(* PLC project SafeLOGIC-1, BrAutomation SafeDESIGNER  5.15.0.0 *)
(* stored: companyURL http://www.br-automation.com, creationDateTime Sun Sep 18 11:29:32 2022 *)

PROGRAM Zone
  VAR  (* added by the conversion: wires and edge detectors of the diagram *)
    _SAFEBOOL_TO_BOOL243_OUT : BOOL;
    _SAFEBOOL_TO_BOOL256_OUT : BOOL;
    _AND_S244_OUT : ANY;
    _BOOL_TO_SAFEBOOL249_OUT : SAFEBOOL;
    _AND_S238_OUT : ANY;
    _OR259_OUT : BOOL;
    _AND246_OUT : BOOL;
  END_VAR

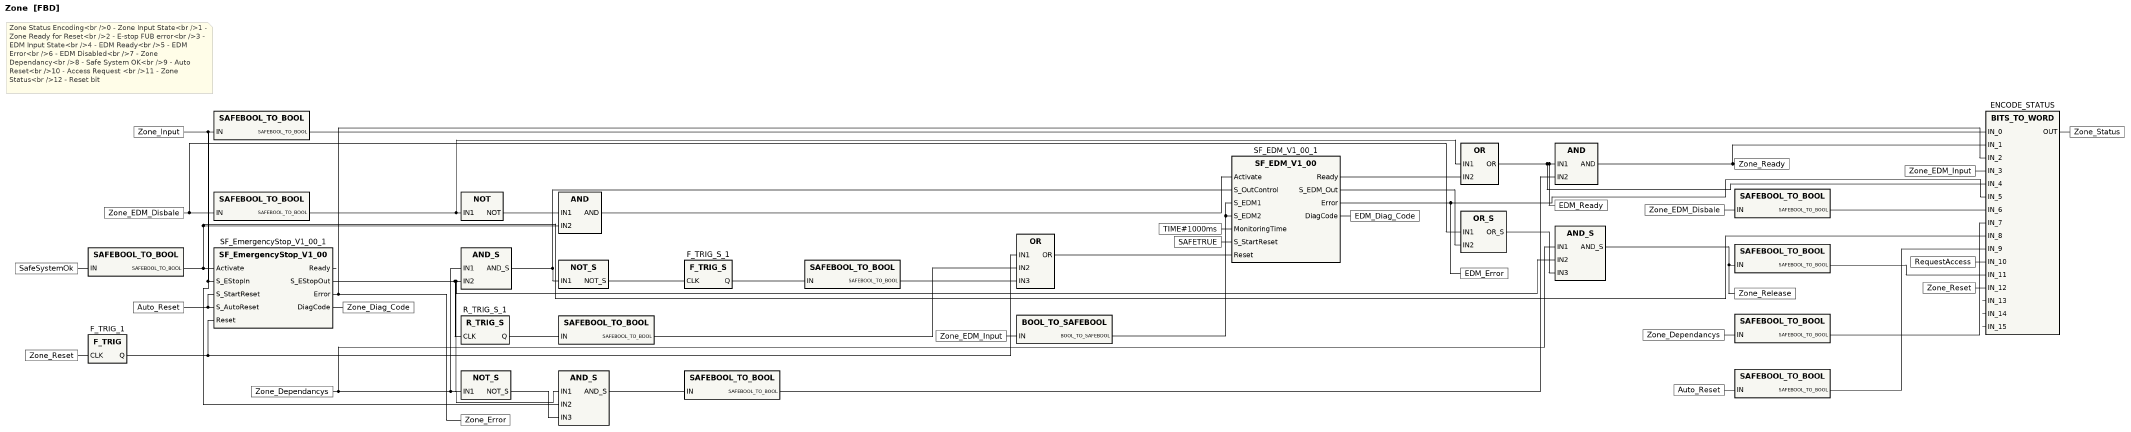
(* FBD diagram, written out as Structured Text *)
_SAFEBOOL_TO_BOOL243_OUT := SAFEBOOL_TO_BOOL(SafeSystemOk);
F_TRIG_1(CLK := Zone_Reset);
SF_EmergencyStop_V1_00_1(Activate := _SAFEBOOL_TO_BOOL243_OUT, S_EStopIn := Zone_Input, S_StartReset := Auto_Reset, S_AutoReset := Auto_Reset, Reset := F_TRIG_1.Q);
_SAFEBOOL_TO_BOOL256_OUT := SAFEBOOL_TO_BOOL(Zone_EDM_Disbale);
_AND_S244_OUT := AND_S(Zone_Dependancys, SF_EmergencyStop_V1_00_1.S_EStopOut);
_BOOL_TO_SAFEBOOL249_OUT := BOOL_TO_SAFEBOOL(Zone_EDM_Input);
R_TRIG_S_1(CLK := SF_EmergencyStop_V1_00_1.S_EStopOut);
F_TRIG_S_1(CLK := NOT_S(_AND_S244_OUT));
SF_EDM_V1_00_1(Activate := NOT _SAFEBOOL_TO_BOOL256_OUT AND _SAFEBOOL_TO_BOOL243_OUT, S_OutControl := _AND_S244_OUT, S_EDM1 := _BOOL_TO_SAFEBOOL249_OUT, S_EDM2 := _BOOL_TO_SAFEBOOL249_OUT, MonitoringTime := TIME#1000ms, S_StartReset := SAFETRUE, Reset := F_TRIG_1.Q OR SAFEBOOL_TO_BOOL(R_TRIG_S_1.Q) OR SAFEBOOL_TO_BOOL(F_TRIG_S_1.Q));
_AND_S238_OUT := AND_S(Zone_Dependancys, SF_EmergencyStop_V1_00_1.S_EStopOut, OR_S(Zone_EDM_Disbale, SF_EDM_V1_00_1.S_EDM_Out));
Zone_Release := _AND_S238_OUT;
EDM_Diag_Code := SF_EDM_V1_00_1.DiagCode;
_OR259_OUT := _SAFEBOOL_TO_BOOL256_OUT OR SF_EDM_V1_00_1.Ready;
EDM_Ready := _OR259_OUT;
EDM_Error := SF_EDM_V1_00_1.Error;
_AND246_OUT := _OR259_OUT AND SAFEBOOL_TO_BOOL(AND_S(Zone_Dependancys, Zone_Input, NOT_S(SF_EmergencyStop_V1_00_1.S_EStopOut)));
Zone_Ready := _AND246_OUT;
Zone_Diag_Code := SF_EmergencyStop_V1_00_1.DiagCode;
Zone_Error := SF_EmergencyStop_V1_00_1.Error;
ENCODE_STATUS(IN_0 := SAFEBOOL_TO_BOOL(Zone_Input), IN_1 := _AND246_OUT, IN_2 := SF_EmergencyStop_V1_00_1.Error, IN_3 := Zone_EDM_Input, IN_4 := _OR259_OUT, IN_5 := SF_EDM_V1_00_1.Error, IN_6 := SAFEBOOL_TO_BOOL(Zone_EDM_Disbale), IN_7 := SAFEBOOL_TO_BOOL(Zone_Dependancys), IN_8 := _SAFEBOOL_TO_BOOL243_OUT, IN_9 := SAFEBOOL_TO_BOOL(Auto_Reset), IN_10 := RequestAccess, IN_11 := SAFEBOOL_TO_BOOL(_AND_S238_OUT), IN_12 := Zone_Reset);
Zone_Status := ENCODE_STATUS.OUT;
(* Zone Status Encoding<br />0 - Zone Input State<br />1 - Zone Ready for Reset<br />2 - E-stop FUB error<br />3 - EDM Input State<br />4 - EDM Ready<br />5 - EDM Error<br />6 - EDM Disabled<br />7 - Zone Dependancy<br />8 - Safe System OK<br />9 - Auto Reset<br />10 - Access Request <br />11 - Zone Status<br />12 - Reset bit *)
END_PROGRAM
